// Mitsubishi GX Works2 project: hello_world   PLC: Q03UDV
// LRI_2023

PROGRAM MAIN
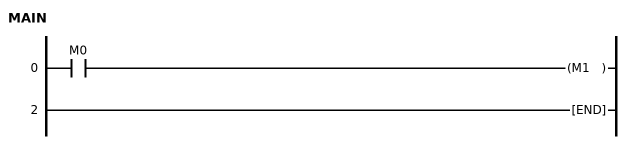
0     LD      M0
      OUT     M1
2     END
END_PROGRAM
